FUNCTION_BLOCK TSV

VAR_INPUT
	IN : BOOL;
	PT : TIME := T#2s;
END_VAR
VAR_OUTPUT
	Q : BOOL;
END_VAR
VAR
	rTrig : R_TRIG;
	tonTime : TON;
	
END_VAR

(*
SV-Verhalten [AWL-SV gibt es in ST nicht, deshalb dieser Nachbau]:
SV <Zeit> startet die adressierte Zeit, wenn das VKE von "0" auf "1" wechselt. Die programmierte
Zeitdauer läuft ab, auch wenn das VKE inzwischen auf "0" wechselt. Wechselt das VKE von "0" auf
"1", bevor die programmierte Zeit abgelaufen ist, wird die programmierte Zeitdauer neu gestartet.
*)

rTrig(CLK := IN);
IF rTrig.Q THEN
	tonTime(IN := FALSE, PT := PT);
	Q := TRUE;
END_IF

tonTime(IN := Q, PT := PT);

IF tonTime.Q THEN
	Q := FALSE;
END_IF

END_FUNCTION_BLOCK

(* stored: Version 1.1.0.1, ProductVersion 3.1.4024.3
   POU TSV: Id {9b44882a-5eda-4ddc-93c2-52d832530036}, SpecialFunc None *)
